KUKA KRL program: td.src, td.dat

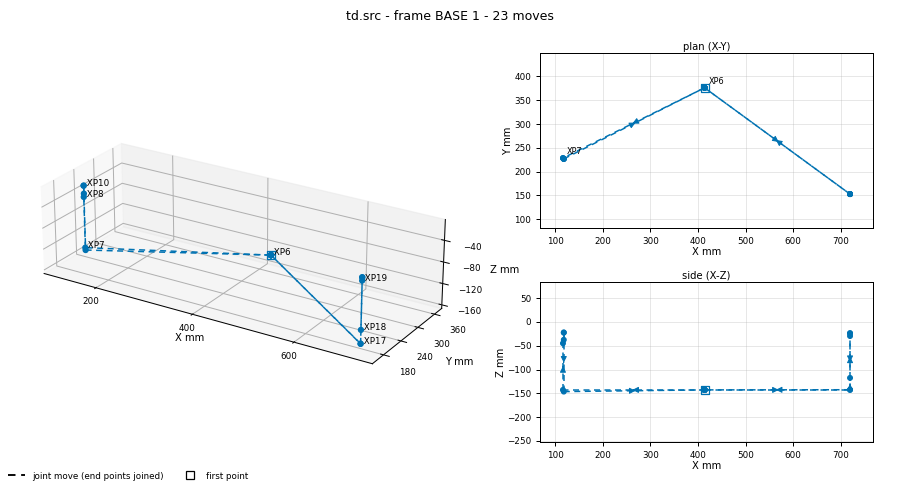
[picture p0: tool path of td.src in frame BASE 1, 23 of 23 moves have a stored position in this frame; points joined in program order, loops and branches not executed]
--- td.src ---
&ACCESS RVO
&REL 27
&PARAM EDITMASK = *
&PARAM TEMPLATE = C:\KRC\Roboter\Template\vorgabe
&PARAM DISKPATH = KRC:\R1\Program\MEEC25\Group3
DEF td( )
;FOLD INI;%{PE}
  ;FOLD BASISTECH INI
    GLOBAL INTERRUPT DECL 3 WHEN $STOPMESS==TRUE DO IR_STOPM ( )
    INTERRUPT ON 3
    BAS (#INITMOV,0 )
  ;ENDFOLD (BASISTECH INI)
  ;FOLD USER INI
    ;Make your modifications here

  ;ENDFOLD (USER INI)
  ;ENDFOLD (INI)
;=======================================================================
;============ Movimento Ponto de Recolha 1 -> Balde Amarelo ============
;=======================================================================
;FOLD PTP P6 Vel=80 % PDAT6 Tool[2]:Tool_G3 Base[1]:Base_G3 ;%{PE}
;FOLD Parameters ;%{h}
;Params IlfProvider=kukaroboter.basistech.inlineforms.movement.old; Kuka.IsGlobalPoint=False; Kuka.PointName=P6; Kuka.BlendingEnabled=False; Kuka.MoveDataPtpName=PDAT6; Kuka.VelocityPtp=80; Kuka.CurrentCDSetIndex=0; Kuka.MovementParameterFieldEnabled=True; IlfCommand=PTP
;ENDFOLD
$BWDSTART = FALSE
PDAT_ACT = PPDAT6
FDAT_ACT = FP6
BAS(#PTP_PARAMS, 80.0)
SET_CD_PARAMS (0)
PTP XP6
;ENDFOLD

;FOLD PTP P7 Vel=80 % PDAT7 Tool[2]:Tool_G3 Base[1]:Base_G3 ;%{PE}
;FOLD Parameters ;%{h}
;Params IlfProvider=kukaroboter.basistech.inlineforms.movement.old; Kuka.IsGlobalPoint=False; Kuka.PointName=P7; Kuka.BlendingEnabled=False; Kuka.MoveDataPtpName=PDAT7; Kuka.VelocityPtp=80; Kuka.CurrentCDSetIndex=0; Kuka.MovementParameterFieldEnabled=True; IlfCommand=PTP
;ENDFOLD
$BWDSTART = FALSE
PDAT_ACT = PPDAT7
FDAT_ACT = FP7
BAS(#PTP_PARAMS, 80.0)
SET_CD_PARAMS (0)
PTP XP7
;ENDFOLD

;FOLD PTP P8 Vel=40 % PDAT8 Tool[2]:Tool_G3 Base[1]:Base_G3 ;%{PE}
;FOLD Parameters ;%{h}
;Params IlfProvider=kukaroboter.basistech.inlineforms.movement.old; Kuka.IsGlobalPoint=False; Kuka.PointName=P8; Kuka.BlendingEnabled=False; Kuka.MoveDataPtpName=PDAT8; Kuka.VelocityPtp=40; Kuka.CurrentCDSetIndex=0; Kuka.MovementParameterFieldEnabled=True; IlfCommand=PTP
;ENDFOLD
$BWDSTART = FALSE
PDAT_ACT = PPDAT8
FDAT_ACT = FP8
BAS(#PTP_PARAMS, 40.0)
SET_CD_PARAMS (0)
PTP XP8
;ENDFOLD

;FOLD PTP P9 Vel=100 % PDAT9 Tool[2]:Tool_G3 Base[1]:Base_G3 ;%{PE}
;FOLD Parameters ;%{h}
;Params IlfProvider=kukaroboter.basistech.inlineforms.movement.old; Kuka.IsGlobalPoint=False; Kuka.PointName=P9; Kuka.BlendingEnabled=False; Kuka.MoveDataPtpName=PDAT9; Kuka.VelocityPtp=100; Kuka.CurrentCDSetIndex=0; Kuka.MovementParameterFieldEnabled=True; IlfCommand=PTP
;ENDFOLD
$BWDSTART = FALSE
PDAT_ACT = PPDAT9
FDAT_ACT = FP9
BAS(#PTP_PARAMS, 100.0)
SET_CD_PARAMS (0)
PTP XP9
;ENDFOLD

;FOLD PTP P10 Vel=50 % PDAT10 Tool[2]:Tool_G3 Base[1]:Base_G3 ;%{PE}
;FOLD Parameters ;%{h}
;Params IlfProvider=kukaroboter.basistech.inlineforms.movement.old; Kuka.IsGlobalPoint=False; Kuka.PointName=P10; Kuka.BlendingEnabled=False; Kuka.MoveDataPtpName=PDAT10; Kuka.VelocityPtp=50; Kuka.CurrentCDSetIndex=0; Kuka.MovementParameterFieldEnabled=True; IlfCommand=PTP
;ENDFOLD
$BWDSTART = FALSE
PDAT_ACT = PPDAT10
FDAT_ACT = FP10
BAS(#PTP_PARAMS, 50.0)
SET_CD_PARAMS (0)
PTP XP10
;ENDFOLD

;FOLD PTP P11 Vel=100 % PDAT11 Tool[2]:Tool_G3 Base[1]:Base_G3 ;%{PE}
;FOLD Parameters ;%{h}
;Params IlfProvider=kukaroboter.basistech.inlineforms.movement.old; Kuka.IsGlobalPoint=False; Kuka.PointName=P11; Kuka.BlendingEnabled=False; Kuka.MoveDataPtpName=PDAT11; Kuka.VelocityPtp=100; Kuka.CurrentCDSetIndex=0; Kuka.MovementParameterFieldEnabled=True; IlfCommand=PTP
;ENDFOLD
$BWDSTART = FALSE
PDAT_ACT = PPDAT11
FDAT_ACT = FP11
BAS(#PTP_PARAMS, 100.0)
SET_CD_PARAMS (0)
PTP XP11
;ENDFOLD

;FOLD PTP P12 Vel=50 % PDAT12 Tool[2]:Tool_G3 Base[1]:Base_G3 ;%{PE}
;FOLD Parameters ;%{h}
;Params IlfProvider=kukaroboter.basistech.inlineforms.movement.old; Kuka.IsGlobalPoint=False; Kuka.PointName=P12; Kuka.BlendingEnabled=False; Kuka.MoveDataPtpName=PDAT12; Kuka.VelocityPtp=50; Kuka.CurrentCDSetIndex=0; Kuka.MovementParameterFieldEnabled=True; IlfCommand=PTP
;ENDFOLD
$BWDSTART = FALSE
PDAT_ACT = PPDAT12
FDAT_ACT = FP12
BAS(#PTP_PARAMS, 50.0)
SET_CD_PARAMS (0)
PTP XP12
;ENDFOLD

;FOLD PTP P14 Vel=80 % PDAT14 Tool[2]:Tool_G3 Base[1]:Base_G3 ;%{PE}
;FOLD Parameters ;%{h}
;Params IlfProvider=kukaroboter.basistech.inlineforms.movement.old; Kuka.IsGlobalPoint=False; Kuka.PointName=P14; Kuka.BlendingEnabled=False; Kuka.MoveDataPtpName=PDAT14; Kuka.VelocityPtp=80; Kuka.CurrentCDSetIndex=0; Kuka.MovementParameterFieldEnabled=True; IlfCommand=PTP
;ENDFOLD
$BWDSTART = FALSE
PDAT_ACT = PPDAT14
FDAT_ACT = FP14
BAS(#PTP_PARAMS, 80.0)
SET_CD_PARAMS (0)
PTP XP14
;ENDFOLD

;FOLD PTP P17 Vel=80 % PDAT17 Tool[2]:Tool_G3 Base[1]:Base_G3 ;%{PE}
;FOLD Parameters ;%{h}
;Params IlfProvider=kukaroboter.basistech.inlineforms.movement.old; Kuka.IsGlobalPoint=False; Kuka.PointName=P17; Kuka.BlendingEnabled=False; Kuka.MoveDataPtpName=PDAT17; Kuka.VelocityPtp=80; Kuka.CurrentCDSetIndex=0; Kuka.MovementParameterFieldEnabled=True; IlfCommand=PTP
;ENDFOLD
$BWDSTART = FALSE
PDAT_ACT = PPDAT17
FDAT_ACT = FP17
BAS(#PTP_PARAMS, 80.0)
SET_CD_PARAMS (0)
PTP XP17
;ENDFOLD

;FOLD PTP P18 Vel=80 % PDAT18 Tool[2]:Tool_G3 Base[1]:Base_G3 ;%{PE}
;FOLD Parameters ;%{h}
;Params IlfProvider=kukaroboter.basistech.inlineforms.movement.old; Kuka.IsGlobalPoint=False; Kuka.PointName=P18; Kuka.BlendingEnabled=False; Kuka.MoveDataPtpName=PDAT18; Kuka.VelocityPtp=80; Kuka.CurrentCDSetIndex=0; Kuka.MovementParameterFieldEnabled=True; IlfCommand=PTP
;ENDFOLD
$BWDSTART = FALSE
PDAT_ACT = PPDAT18
FDAT_ACT = FP18
BAS(#PTP_PARAMS, 80.0)
SET_CD_PARAMS (0)
PTP XP18
;ENDFOLD

;FOLD PTP P19 Vel=80 % PDAT19 Tool[2]:Tool_G3 Base[1]:Base_G3 ;%{PE}
;FOLD Parameters ;%{h}
;Params IlfProvider=kukaroboter.basistech.inlineforms.movement.old; Kuka.IsGlobalPoint=False; Kuka.PointName=P19; Kuka.BlendingEnabled=False; Kuka.MoveDataPtpName=PDAT19; Kuka.VelocityPtp=80; Kuka.CurrentCDSetIndex=0; Kuka.MovementParameterFieldEnabled=True; IlfCommand=PTP
;ENDFOLD
$BWDSTART = FALSE
PDAT_ACT = PPDAT19
FDAT_ACT = FP19
BAS(#PTP_PARAMS, 80.0)
SET_CD_PARAMS (0)
PTP XP19
;ENDFOLD

;FOLD PTP P20 Vel=80 % PDAT20 Tool[2]:Tool_G3 Base[1]:Base_G3 ;%{PE}
;FOLD Parameters ;%{h}
;Params IlfProvider=kukaroboter.basistech.inlineforms.movement.old; Kuka.IsGlobalPoint=False; Kuka.PointName=P20; Kuka.BlendingEnabled=False; Kuka.MoveDataPtpName=PDAT20; Kuka.VelocityPtp=80; Kuka.CurrentCDSetIndex=0; Kuka.MovementParameterFieldEnabled=True; IlfCommand=PTP
;ENDFOLD
$BWDSTART = FALSE
PDAT_ACT = PPDAT20
FDAT_ACT = FP20
BAS(#PTP_PARAMS, 80.0)
SET_CD_PARAMS (0)
PTP XP20
;ENDFOLD

;FOLD PTP P21 Vel=80 % PDAT21 Tool[2]:Tool_G3 Base[1]:Base_G3 ;%{PE}
;FOLD Parameters ;%{h}
;Params IlfProvider=kukaroboter.basistech.inlineforms.movement.old; Kuka.IsGlobalPoint=False; Kuka.PointName=P21; Kuka.BlendingEnabled=False; Kuka.MoveDataPtpName=PDAT21; Kuka.VelocityPtp=80; Kuka.CurrentCDSetIndex=0; Kuka.MovementParameterFieldEnabled=True; IlfCommand=PTP
;ENDFOLD
$BWDSTART = FALSE
PDAT_ACT = PPDAT21
FDAT_ACT = FP21
BAS(#PTP_PARAMS, 80.0)
SET_CD_PARAMS (0)
PTP XP21
;ENDFOLD

;FOLD PTP P22 Vel=80 % PDAT22 Tool[2]:Tool_G3 Base[1]:Base_G3 ;%{PE}
;FOLD Parameters ;%{h}
;Params IlfProvider=kukaroboter.basistech.inlineforms.movement.old; Kuka.IsGlobalPoint=False; Kuka.PointName=P22; Kuka.BlendingEnabled=False; Kuka.MoveDataPtpName=PDAT22; Kuka.VelocityPtp=80; Kuka.CurrentCDSetIndex=0; Kuka.MovementParameterFieldEnabled=True; IlfCommand=PTP
;ENDFOLD
$BWDSTART = FALSE
PDAT_ACT = PPDAT22
FDAT_ACT = FP22
BAS(#PTP_PARAMS, 80.0)
SET_CD_PARAMS (0)
PTP XP22
;ENDFOLD

;FOLD PTP P23 Vel=80 % PDAT23 Tool[2]:Tool_G3 Base[1]:Base_G3 ;%{PE}
;FOLD Parameters ;%{h}
;Params IlfProvider=kukaroboter.basistech.inlineforms.movement.old; Kuka.IsGlobalPoint=False; Kuka.PointName=P23; Kuka.BlendingEnabled=False; Kuka.MoveDataPtpName=PDAT23; Kuka.VelocityPtp=80; Kuka.CurrentCDSetIndex=0; Kuka.MovementParameterFieldEnabled=True; IlfCommand=PTP
;ENDFOLD
$BWDSTART = FALSE
PDAT_ACT = PPDAT23
FDAT_ACT = FP23
BAS(#PTP_PARAMS, 80.0)
SET_CD_PARAMS (0)
PTP XP23
;ENDFOLD

;===================================================================
;========== Movimento Ponto de Recolha 1 -> Balde Verde ============
;===================================================================

;FOLD PTP P25 Vel=80 % PDAT25 Tool[2]:Tool_G3 Base[1]:Base_G3 ;%{PE}
;FOLD Parameters ;%{h}
;Params IlfProvider=kukaroboter.basistech.inlineforms.movement.old; Kuka.IsGlobalPoint=False; Kuka.PointName=P25; Kuka.BlendingEnabled=False; Kuka.MoveDataPtpName=PDAT25; Kuka.VelocityPtp=80; Kuka.CurrentCDSetIndex=0; Kuka.MovementParameterFieldEnabled=True; IlfCommand=PTP
;ENDFOLD
$BWDSTART = FALSE
PDAT_ACT = PPDAT25
FDAT_ACT = FP25
BAS(#PTP_PARAMS, 80.0)
SET_CD_PARAMS (0)
PTP XP25
;ENDFOLD


;=================================================================
;========= Movimento Ponto de Recolha 1 -> Balde Azul ============
;=================================================================

;FOLD PTP P26 Vel=80 % PDAT26 Tool[2]:Tool_G3 Base[1]:Base_G3 ;%{PE}
;FOLD Parameters ;%{h}
;Params IlfProvider=kukaroboter.basistech.inlineforms.movement.old; Kuka.IsGlobalPoint=False; Kuka.PointName=P26; Kuka.BlendingEnabled=False; Kuka.MoveDataPtpName=PDAT26; Kuka.VelocityPtp=80; Kuka.CurrentCDSetIndex=0; Kuka.MovementParameterFieldEnabled=True; IlfCommand=PTP
;ENDFOLD
$BWDSTART = FALSE
PDAT_ACT = PPDAT26
FDAT_ACT = FP26
BAS(#PTP_PARAMS, 80.0)
SET_CD_PARAMS (0)
PTP XP26
;ENDFOLD


;=======================================================================
;============ Movimento Ponto de Recolha 2 -> Balde Amarelo ============
;=======================================================================

;FOLD PTP P27 Vel=80 % PDAT27 Tool[2]:Tool_G3 Base[1]:Base_G3 ;%{PE}
;FOLD Parameters ;%{h}
;Params IlfProvider=kukaroboter.basistech.inlineforms.movement.old; Kuka.IsGlobalPoint=False; Kuka.PointName=P27; Kuka.BlendingEnabled=False; Kuka.MoveDataPtpName=PDAT27; Kuka.VelocityPtp=80; Kuka.CurrentCDSetIndex=0; Kuka.MovementParameterFieldEnabled=True; IlfCommand=PTP
;ENDFOLD
$BWDSTART = FALSE
PDAT_ACT = PPDAT27
FDAT_ACT = FP27
BAS(#PTP_PARAMS, 80.0)
SET_CD_PARAMS (0)
PTP XP27
;ENDFOLD


;===================================================================
;========== Movimento Ponto de Recolha 2 -> Balde Verde ============
;===================================================================

;FOLD PTP P28 Vel=80 % PDAT28 Tool[2]:Tool_G3 Base[1]:Base_G3 ;%{PE}
;FOLD Parameters ;%{h}
;Params IlfProvider=kukaroboter.basistech.inlineforms.movement.old; Kuka.IsGlobalPoint=False; Kuka.PointName=P28; Kuka.BlendingEnabled=False; Kuka.MoveDataPtpName=PDAT28; Kuka.VelocityPtp=80; Kuka.CurrentCDSetIndex=0; Kuka.MovementParameterFieldEnabled=True; IlfCommand=PTP
;ENDFOLD
$BWDSTART = FALSE
PDAT_ACT = PPDAT28
FDAT_ACT = FP28
BAS(#PTP_PARAMS, 80.0)
SET_CD_PARAMS (0)
PTP XP28
;ENDFOLD


;=================================================================
;========= Movimento Ponto de Recolha 2 -> Balde Azul ============
;=================================================================

;FOLD PTP P29 Vel=80 % PDAT29 Tool[2]:Tool_G3 Base[1]:Base_G3 ;%{PE}
;FOLD Parameters ;%{h}
;Params IlfProvider=kukaroboter.basistech.inlineforms.movement.old; Kuka.IsGlobalPoint=False; Kuka.PointName=P29; Kuka.BlendingEnabled=False; Kuka.MoveDataPtpName=PDAT29; Kuka.VelocityPtp=80; Kuka.CurrentCDSetIndex=0; Kuka.MovementParameterFieldEnabled=True; IlfCommand=PTP
;ENDFOLD
$BWDSTART = FALSE
PDAT_ACT = PPDAT29
FDAT_ACT = FP29
BAS(#PTP_PARAMS, 80.0)
SET_CD_PARAMS (0)
PTP XP29
;ENDFOLD


;=======================================================================
;============ Movimento Ponto de Recolha 3 -> Balde Amarelo ============
;=======================================================================

;FOLD PTP P30 Vel=80 % PDAT30 Tool[2]:Tool_G3 Base[1]:Base_G3 ;%{PE}
;FOLD Parameters ;%{h}
;Params IlfProvider=kukaroboter.basistech.inlineforms.movement.old; Kuka.IsGlobalPoint=False; Kuka.PointName=P30; Kuka.BlendingEnabled=False; Kuka.MoveDataPtpName=PDAT30; Kuka.VelocityPtp=80; Kuka.CurrentCDSetIndex=0; Kuka.MovementParameterFieldEnabled=True; IlfCommand=PTP
;ENDFOLD
$BWDSTART = FALSE
PDAT_ACT = PPDAT30
FDAT_ACT = FP30
BAS(#PTP_PARAMS, 80.0)
SET_CD_PARAMS (0)
PTP XP30
;ENDFOLD


;===================================================================
;========== Movimento Ponto de Recolha 3 -> Balde Verde ============
;===================================================================

;FOLD PTP P31 Vel=80 % PDAT31 Tool[2]:Tool_G3 Base[1]:Base_G3 ;%{PE}
;FOLD Parameters ;%{h}
;Params IlfProvider=kukaroboter.basistech.inlineforms.movement.old; Kuka.IsGlobalPoint=False; Kuka.PointName=P31; Kuka.BlendingEnabled=False; Kuka.MoveDataPtpName=PDAT31; Kuka.VelocityPtp=80; Kuka.CurrentCDSetIndex=0; Kuka.MovementParameterFieldEnabled=True; IlfCommand=PTP
;ENDFOLD
$BWDSTART = FALSE
PDAT_ACT = PPDAT31
FDAT_ACT = FP31
BAS(#PTP_PARAMS, 80.0)
SET_CD_PARAMS (0)
PTP XP31
;ENDFOLD


;=================================================================
;========= Movimento Ponto de Recolha 3 -> Balde Azul ============
;=================================================================

;FOLD PTP P32 Vel=80 % PDAT32 Tool[2]:Tool_G3 Base[1]:Base_G3 ;%{PE}
;FOLD Parameters ;%{h}
;Params IlfProvider=kukaroboter.basistech.inlineforms.movement.old; Kuka.IsGlobalPoint=False; Kuka.PointName=P32; Kuka.BlendingEnabled=False; Kuka.MoveDataPtpName=PDAT32; Kuka.VelocityPtp=80; Kuka.CurrentCDSetIndex=0; Kuka.MovementParameterFieldEnabled=True; IlfCommand=PTP
;ENDFOLD
$BWDSTART = FALSE
PDAT_ACT = PPDAT32
FDAT_ACT = FP32
BAS(#PTP_PARAMS, 80.0)
SET_CD_PARAMS (0)
PTP XP32
;ENDFOLD


END

--- td.dat ---
&ACCESS RVP
&REL 26
&PARAM EDITMASK = *
&PARAM TEMPLATE = C:\KRC\Roboter\Template\vorgabe
&PARAM DISKPATH = KRC:\R1\Program\MEEC25\Group3
DEFDAT  TD
;FOLD EXTERNAL DECLARATIONS;%{PE}%MKUKATPBASIS,%CEXT,%VCOMMON,%P
;FOLD BASISTECH EXT;%{PE}%MKUKATPBASIS,%CEXT,%VEXT,%P
EXT  BAS (BAS_COMMAND  :IN,REAL  :IN )
DECL INT SUCCESS
;ENDFOLD (BASISTECH EXT)
;FOLD USER EXT;%{E}%MKUKATPUSER,%CEXT,%VEXT,%P
;Make your modifications here

;ENDFOLD (USER EXT)
;ENDFOLD (EXTERNAL DECLARATIONS)
DECL E6POS XP1={X 499.803619,Y 13.5229921,Z 160.789398,A 0.0,B 90.0000,C -86.9811096,S 2,T 8,E1 0.0,E2 0.0,E3 0.0,E4 0.0,E5 0.0,E6 0.0}
DECL FDAT FP1={TOOL_NO 1,BASE_NO 0,IPO_FRAME #BASE,POINT2[] " "}
DECL PDAT PPDAT1={VEL 50.0000,ACC 100.000,APO_DIST 500.000,APO_MODE #CDIS,GEAR_JERK 100.000,EXAX_IGN 0}
DECL MODULEPARAM_T LAST_TP_PARAMS={PARAMS[] "Kuka.VelocityFieldEnabled=True; Kuka.ColDetectFieldEnabled=True; Kuka.MovementParameterFieldEnabled=True; Kuka.IsAngleEnabled=False; Kuka.PointName=P22; Kuka.FrameData.base_no=1; Kuka.FrameData.tool_no=2; Kuka.FrameData.ipo_frame=#BASE; Kuka.isglobalpoint=False; Kuka.MoveDataPtpName=PDAT22; Kuka.MovementDataPdat.apo_mode=#CDIS; Kuka.MovementDataPdat.apo_dist=500; Kuka.MovementData.vel=80; Kuka.MovementData.acc=100; Kuka.MovementData.exax_ign=0; Kuka.VelocityPtp=80; Kuka.BlendingEnabled=False; Kuka.APXEnabled=False; Kuka.CurrentCDSetIndex=0; Kuka.FrameData.point2=  "}
DECL E6POS XP2={X 348.651459,Y -280.706909,Z 106.842758,A 0.0,B 90.0000,C -21.4602699,S 0,T 11,E1 0.0,E2 0.0,E3 0.0,E4 0.0,E5 0.0,E6 0.0}
DECL FDAT FP2={TOOL_NO 1,BASE_NO 0,IPO_FRAME #BASE,POINT2[] " "}
DECL PDAT PPDAT2={VEL 50.0000,ACC 100.000,APO_DIST 500.000,APO_MODE #CDIS,GEAR_JERK 100.000,EXAX_IGN 0}
DECL E6POS XP3={X 348.651459,Y -280.706909,Z 56.8600044,A 0.0,B 90.0000,C -21.4602699,S 0,T 11,E1 0.0,E2 0.0,E3 0.0,E4 0.0,E5 0.0,E6 0.0}
DECL FDAT FP3={TOOL_NO 1,BASE_NO 0,IPO_FRAME #BASE,POINT2[] " "}
DECL PDAT PPDAT3={VEL 50.0000,ACC 100.000,APO_DIST 500.000,APO_MODE #CDIS,GEAR_JERK 100.000,EXAX_IGN 0}
DECL E6POS XP4={X 348.651459,Y -280.706909,Z 56.8600044,A 0.0,B 90.0000,C -64.5600052,S 0,T 11,E1 0.0,E2 0.0,E3 0.0,E4 0.0,E5 0.0,E6 0.0}
DECL FDAT FP4={TOOL_NO 2,BASE_NO 1,IPO_FRAME #BASE,POINT2[] " "}
DECL PDAT PPDAT4={VEL 50.0000,ACC 100.000,APO_DIST 500.000,APO_MODE #CDIS,GEAR_JERK 100.000,EXAX_IGN 0}
DECL E6POS XP5={X 499.803619,Y 13.5229921,Z 160.789398,A 0.0,B 90.0000,C -86.9811096,S 2,T 8,E1 0.0,E2 0.0,E3 0.0,E4 0.0,E5 0.0,E6 0.0}
DECL FDAT FP5={TOOL_NO 1,BASE_NO 0,IPO_FRAME #BASE,POINT2[] " "}
DECL PDAT PPDAT5={VEL 50.0000,ACC 100.000,APO_DIST 500.000,APO_MODE #CDIS,GEAR_JERK 100.000,EXAX_IGN 0}
DECL E6POS XP6={X 413.672638,Y 376.212982,Z -142.734314,A 0.0,B -90.0000,C 2.66616058,S 2,T 8,E1 0.0,E2 0.0,E3 0.0,E4 0.0,E5 0.0,E6 0.0}
DECL FDAT FP6={TOOL_NO 2,BASE_NO 1,IPO_FRAME #BASE,POINT2[] " "}
DECL PDAT PPDAT6={VEL 80.0000,ACC 100.000,APO_DIST 500.000,APO_MODE #CDIS,GEAR_JERK 100.000,EXAX_IGN 0}
DECL E6POS XP7={X 116.247948,Y 228.584106,Z -142.734314,A 0.0,B -90.0000,C 66.6335373,S 0,T 11,E1 0.0,E2 0.0,E3 0.0,E4 0.0,E5 0.0,E6 0.0}
DECL FDAT FP7={TOOL_NO 2,BASE_NO 1,IPO_FRAME #BASE,POINT2[] " "}
DECL PDAT PPDAT7={VEL 80.0000,ACC 100.000,APO_DIST 500.000,APO_MODE #CDIS,GEAR_JERK 100.000,EXAX_IGN 0}
DECL E6POS XP8={X 116.247948,Y 228.584106,Z -44.8425179,A 0.0,B -90.0000,C 66.2220306,S 0,T 11,E1 0.0,E2 0.0,E3 0.0,E4 0.0,E5 0.0,E6 0.0}
DECL FDAT FP8={TOOL_NO 2,BASE_NO 1,IPO_FRAME #BASE,POINT2[] " "}
DECL PDAT PPDAT8={VEL 40.0000,ACC 100.000,APO_DIST 500.000,APO_MODE #CDIS,GEAR_JERK 100.000,EXAX_IGN 0}
DECL E6POS XP9={X 117.963219,Y 226.885269,Z -37.4893417,A 0.0,B -90.0000,C 142.230179,S 0,T 11,E1 0.0,E2 0.0,E3 0.0,E4 0.0,E5 0.0,E6 0.0}
DECL FDAT FP9={TOOL_NO 2,BASE_NO 1,IPO_FRAME #BASE,POINT2[] " "}
DECL PDAT PPDAT9={VEL 100.000,ACC 100.000,APO_DIST 500.000,APO_MODE #CDIS,GEAR_JERK 100.000,EXAX_IGN 0}
DECL E6POS XP10={X 117.963219,Y 226.885269,Z -22.2715874,A 0.0,B -90.0000,C 142.230179,S 0,T 11,E1 0.0,E2 0.0,E3 0.0,E4 0.0,E5 0.0,E6 0.0}
DECL FDAT FP10={TOOL_NO 2,BASE_NO 1,IPO_FRAME #BASE,POINT2[] " "}
DECL PDAT PPDAT10={VEL 50.0000,ACC 100.000,APO_DIST 500.000,APO_MODE #CDIS,GEAR_JERK 100.000,EXAX_IGN 0}
DECL E6POS XP11={X 117.963219,Y 226.885269,Z -22.2715874,A 0.0,B -90.0000,C 81.6844330,S 0,T 11,E1 0.0,E2 0.0,E3 0.0,E4 0.0,E5 0.0,E6 0.0}
DECL FDAT FP11={TOOL_NO 2,BASE_NO 1,IPO_FRAME #BASE,POINT2[] " "}
DECL PDAT PPDAT11={VEL 100.000,ACC 100.000,APO_DIST 500.000,APO_MODE #CDIS,GEAR_JERK 100.000,EXAX_IGN 0}
DECL E6POS XP12={X 117.963219,Y 226.885269,Z -146.318817,A 0.0,B -90.0000,C 81.6844330,S 0,T 11,E1 0.0,E2 0.0,E3 0.0,E4 0.0,E5 0.0,E6 0.0}
DECL FDAT FP12={TOOL_NO 2,BASE_NO 1,IPO_FRAME #BASE,POINT2[] " "}
DECL PDAT PPDAT12={VEL 50.0000,ACC 100.000,APO_DIST 500.000,APO_MODE #CDIS,GEAR_JERK 100.000,EXAX_IGN 0}
DECL E6POS XP13={X 413.672638,Y 376.212982,Z -142.734314,A 0.0,B -90.0000,C 2.66616058,S 2,T 8,E1 0.0,E2 0.0,E3 0.0,E4 0.0,E5 0.0,E6 0.0}
DECL FDAT FP13={TOOL_NO 2,BASE_NO 1,IPO_FRAME #BASE,POINT2[] " "}
DECL PDAT PPDAT13={VEL 50.0000,ACC 100.000,APO_DIST 500.000,APO_MODE #CDIS,GEAR_JERK 100.000,EXAX_IGN 0}
DECL E6POS XP14={X 413.672638,Y 376.212982,Z -142.734314,A 0.0,B -90.0000,C 2.66616058,S 2,T 8,E1 0.0,E2 0.0,E3 0.0,E4 0.0,E5 0.0,E6 0.0}
DECL FDAT FP14={TOOL_NO 2,BASE_NO 1,IPO_FRAME #BASE,POINT2[] " "}
DECL PDAT PPDAT14={VEL 80.0000,ACC 100.000,APO_DIST 500.000,APO_MODE #CDIS,GEAR_JERK 100.000,EXAX_IGN 0}
DECL E6POS XP15={X 717.035,Y 154.325989,Z -143.451050,A 0.0,B -90.0000,C -95.9614182,S 2,T 8,E1 0.0,E2 0.0,E3 0.0,E4 0.0,E5 0.0,E6 0.0}
DECL FDAT FP15={TOOL_NO 2,BASE_NO 1,IPO_FRAME #BASE,POINT2[] " "}
DECL PDAT PPDAT15={VEL 80.0000,ACC 100.000,APO_DIST 500.000,APO_MODE #CDIS,GEAR_JERK 100.000,EXAX_IGN 0}
DECL E6POS XP16={X 716.455322,Y 154.329071,Z -21.3514309,A 0.0,B -90.0000,C -95.6490250,S 2,T 8,E1 0.0,E2 0.0,E3 0.0,E4 0.0,E5 0.0,E6 0.0}
DECL FDAT FP16={TOOL_NO 2,BASE_NO 1,IPO_FRAME #BASE,POINT2[] " "}
DECL PDAT PPDAT16={VEL 80.0000,ACC 100.000,APO_DIST 500.000,APO_MODE #CDIS,GEAR_JERK 100.000,EXAX_IGN 0}
DECL E6POS XP17={X 719.244507,Y 152.886154,Z -142.734314,A 0.0,B -90.0000,C -97.5447083,S 2,T 8,E1 0.0,E2 0.0,E3 0.0,E4 0.0,E5 0.0,E6 0.0}
DECL FDAT FP17={TOOL_NO 2,BASE_NO 1,IPO_FRAME #BASE,POINT2[] " "}
DECL PDAT PPDAT17={VEL 80.0000,ACC 100.000,APO_DIST 500.000,APO_MODE #CDIS,GEAR_JERK 100.000,EXAX_IGN 0}
DECL E6POS XP18={X 719.244507,Y 152.886154,Z -117.521515,A 0.0,B -90.0000,C -97.5447083,S 2,T 8,E1 0.0,E2 0.0,E3 0.0,E4 0.0,E5 0.0,E6 0.0}
DECL FDAT FP18={TOOL_NO 2,BASE_NO 1,IPO_FRAME #BASE,POINT2[] " "}
DECL PDAT PPDAT18={VEL 80.0000,ACC 100.000,APO_DIST 500.000,APO_MODE #CDIS,GEAR_JERK 100.000,EXAX_IGN 0}
DECL E6POS XP19={X 719.244507,Y 152.886154,Z -29.5992737,A 0.0,B -90.0000,C -97.5447083,S 2,T 8,E1 0.0,E2 0.0,E3 0.0,E4 0.0,E5 0.0,E6 0.0}
DECL FDAT FP19={TOOL_NO 2,BASE_NO 1,IPO_FRAME #BASE,POINT2[] " "}
DECL PDAT PPDAT19={VEL 80.0000,ACC 100.000,APO_DIST 500.000,APO_MODE #CDIS,GEAR_JERK 100.000,EXAX_IGN 0}
DECL E6POS XP20={X 719.244507,Y 152.886154,Z -23.7054768,A 0.0,B -90.0000,C -97.5447083,S 2,T 8,E1 0.0,E2 0.0,E3 0.0,E4 0.0,E5 0.0,E6 0.0}
DECL FDAT FP20={TOOL_NO 2,BASE_NO 1,IPO_FRAME #BASE,POINT2[] " "}
DECL PDAT PPDAT20={VEL 80.0000,ACC 100.000,APO_DIST 500.000,APO_MODE #CDIS,GEAR_JERK 100.000,EXAX_IGN 0}
DECL E6POS XP21={X 719.244507,Y 152.886154,Z -23.7054768,A 0.0,B -90.0000,C -158.041901,S 2,T 8,E1 0.0,E2 0.0,E3 0.0,E4 0.0,E5 0.0,E6 0.0}
DECL FDAT FP21={TOOL_NO 2,BASE_NO 1,IPO_FRAME #BASE,POINT2[] " "}
DECL PDAT PPDAT21={VEL 80.0000,ACC 100.000,APO_DIST 500.000,APO_MODE #CDIS,GEAR_JERK 100.000,EXAX_IGN 0}
DECL E6POS XP22={X 719.244507,Y 152.886154,Z -142.380447,A 0.0,B -90.0000,C -158.041901,S 2,T 8,E1 0.0,E2 0.0,E3 0.0,E4 0.0,E5 0.0,E6 0.0}
DECL FDAT FP22={TOOL_NO 2,BASE_NO 1,IPO_FRAME #BASE,POINT2[] " "}
DECL PDAT PPDAT22={VEL 80.0000,ACC 100.000,APO_DIST 500.000,APO_MODE #CDIS,GEAR_JERK 100.000,EXAX_IGN 0}
DECL E6POS XP23={X 413.672638,Y 376.212982,Z -142.734314,A 0.0,B -90.0000,C 2.66616058,S 2,T 8,E1 0.0,E2 0.0,E3 0.0,E4 0.0,E5 0.0,E6 0.0}
DECL FDAT FP23={TOOL_NO 2,BASE_NO 1,IPO_FRAME #BASE,POINT2[] " "}
DECL PDAT PPDAT23={VEL 80.0000,ACC 100.000,APO_DIST 500.000,APO_MODE #CDIS,GEAR_JERK 100.000,EXAX_IGN 0}
DECL E6POS XP24={X 413.672638,Y 376.212982,Z -142.734314,A 0.0,B -90.0000,C 2.66616058,S 2,T 8,E1 0.0,E2 0.0,E3 0.0,E4 0.0,E5 0.0,E6 0.0}
DECL FDAT FP24={TOOL_NO 2,BASE_NO 1,IPO_FRAME #BASE,POINT2[] " "}
DECL PDAT PPDAT24={VEL 80.0000,ACC 100.000,APO_DIST 500.000,APO_MODE #CDIS,GEAR_JERK 100.000,EXAX_IGN 0}
DECL E6POS XP25={X 413.672638,Y 376.212982,Z -142.734314,A 0.0,B -90.0000,C 2.66616058,S 2,T 8,E1 0.0,E2 0.0,E3 0.0,E4 0.0,E5 0.0,E6 0.0}
DECL FDAT FP25={TOOL_NO 2,BASE_NO 1,IPO_FRAME #BASE,POINT2[] " "}
DECL PDAT PPDAT25={VEL 80.0000,ACC 100.000,APO_DIST 500.000,APO_MODE #CDIS,GEAR_JERK 100.000,EXAX_IGN 0}
DECL E6POS XP26={X 413.672638,Y 376.212982,Z -142.734314,A 0.0,B -90.0000,C 2.66616058,S 2,T 8,E1 0.0,E2 0.0,E3 0.0,E4 0.0,E5 0.0,E6 0.0}
DECL FDAT FP26={TOOL_NO 2,BASE_NO 1,IPO_FRAME #BASE,POINT2[] " "}
DECL PDAT PPDAT26={VEL 80.0000,ACC 100.000,APO_DIST 500.000,APO_MODE #CDIS,GEAR_JERK 100.000,EXAX_IGN 0}
DECL E6POS XP27={X 413.672638,Y 376.212982,Z -142.734314,A 0.0,B -90.0000,C 2.66616058,S 2,T 8,E1 0.0,E2 0.0,E3 0.0,E4 0.0,E5 0.0,E6 0.0}
DECL FDAT FP27={TOOL_NO 2,BASE_NO 1,IPO_FRAME #BASE,POINT2[] " "}
DECL PDAT PPDAT27={VEL 80.0000,ACC 100.000,APO_DIST 500.000,APO_MODE #CDIS,GEAR_JERK 100.000,EXAX_IGN 0}
DECL E6POS XP28={X 413.672638,Y 376.212982,Z -142.734314,A 0.0,B -90.0000,C 2.66616058,S 2,T 8,E1 0.0,E2 0.0,E3 0.0,E4 0.0,E5 0.0,E6 0.0}
DECL FDAT FP28={TOOL_NO 2,BASE_NO 1,IPO_FRAME #BASE,POINT2[] " "}
DECL PDAT PPDAT28={VEL 80.0000,ACC 100.000,APO_DIST 500.000,APO_MODE #CDIS,GEAR_JERK 100.000,EXAX_IGN 0}
DECL E6POS XP29={X 413.672638,Y 376.212982,Z -142.734314,A 0.0,B -90.0000,C 2.66616058,S 2,T 8,E1 0.0,E2 0.0,E3 0.0,E4 0.0,E5 0.0,E6 0.0}
DECL FDAT FP29={TOOL_NO 2,BASE_NO 1,IPO_FRAME #BASE,POINT2[] " "}
DECL PDAT PPDAT29={VEL 80.0000,ACC 100.000,APO_DIST 500.000,APO_MODE #CDIS,GEAR_JERK 100.000,EXAX_IGN 0}
DECL E6POS XP30={X 413.672638,Y 376.212982,Z -142.734314,A 0.0,B -90.0000,C 2.66616058,S 2,T 8,E1 0.0,E2 0.0,E3 0.0,E4 0.0,E5 0.0,E6 0.0}
DECL FDAT FP30={TOOL_NO 2,BASE_NO 1,IPO_FRAME #BASE,POINT2[] " "}
DECL PDAT PPDAT30={VEL 80.0000,ACC 100.000,APO_DIST 500.000,APO_MODE #CDIS,GEAR_JERK 100.000,EXAX_IGN 0}
DECL E6POS XP31={X 413.672638,Y 376.212982,Z -142.734314,A 0.0,B -90.0000,C 2.66616058,S 2,T 8,E1 0.0,E2 0.0,E3 0.0,E4 0.0,E5 0.0,E6 0.0}
DECL FDAT FP31={TOOL_NO 2,BASE_NO 1,IPO_FRAME #BASE,POINT2[] " "}
DECL PDAT PPDAT31={VEL 80.0000,ACC 100.000,APO_DIST 500.000,APO_MODE #CDIS,GEAR_JERK 100.000,EXAX_IGN 0}
DECL E6POS XP32={X 413.672638,Y 376.212982,Z -142.734314,A 0.0,B -90.0000,C 2.66616058,S 2,T 8,E1 0.0,E2 0.0,E3 0.0,E4 0.0,E5 0.0,E6 0.0}
DECL FDAT FP32={TOOL_NO 2,BASE_NO 1,IPO_FRAME #BASE,POINT2[] " "}
DECL PDAT PPDAT32={VEL 80.0000,ACC 100.000,APO_DIST 500.000,APO_MODE #CDIS,GEAR_JERK 100.000,EXAX_IGN 0}
ENDDAT
